// TIA Portal project "FuncionFC" (V16)

(* hardware
DEVICE "S7-1200 station_1"  S7-1200 Station
   slot 0: "Rack_0"  S7-1200 Rack  Rack  V1.0
   slot 1: "PLC_1"  CPU 1214C AC/DC/Rly  6ES7 214-1BG40-0XB0  V4.4
*)

// ===== PLC "PLC_1"  CPU 1214C AC/DC/Rly =====

VAR_GLOBAL   // PLC tag table "Tabla de variables estándar"
   ""START"" AT %I0.0 : Bool;
   ""S A"" AT %I0.1 : Bool;
   ""S B"" AT %I0.2 : Bool;
   ""S C"" AT %I0.3 : Bool;
   ""S D"" AT %I0.4 : Bool;
   ""S AB"" AT %I0.5 : Bool;
   ""S CD"" AT %I0.6 : Bool;
   ""S ABCD"" AT %I0.7 : Bool;
   ""EV A"" AT %Q1.0 : Bool;
   ""EV B"" AT %Q1.1 : Bool;
   ""EV C"" AT %Q1.2 : Bool;
   ""EV D"" AT %Q1.3 : Bool;
   ""EV AB"" AT %Q1.4 : Bool;
   ""EV DC"" AT %Q1.5 : Bool;
   ""EV ABCD"" AT %Q1.6 : Bool;
END_VAR